FUNCTION_BLOCK FB_Cylinder EXTENDS FB_Component
VAR_INPUT
END_VAR
VAR_OUTPUT
END_VAR
VAR
	bInputA					AT%I*:		BOOL;
	bInputB					AT%I*:		BOOL;
	bOutputA				AT%Q*:		BOOL;
	bOutputB				AT%Q*:		BOOL;
	stSettings:				ST_CylinderSettings;
	fbDebounceA:			FB_Debounce;
	fbDebounceB:			FB_Debounce;	
	fbTimeout:				TON;
END_VAR

METHOD PUBLIC M_Cycle
VAR_INPUT
END_VAR
SUPER^.M_Cycle();

// Timeout
fbTimeout();
fbTimeout.IN:= FALSE;

// Debounc inputs
fbDebounceA(bInput:= bInputA);
fbDebounceB(bInput:= bInputB);
END_METHOD

METHOD PUBLIC M_Disable : BOOL
VAR_INPUT
END_VAR
bOutputA:= FALSE;
bOutputB:= FALSE;
M_Disable:= TRUE;
END_METHOD

METHOD PROTECTED M_Execute : BOOL // Return state complete
VAR_INPUT
END_VAR
IF M_HasMode(E_Mode.Manual) OR Globals.bSimulation THEN
	;
ELSE
	IF fbDebounceA.bValue AND fbDebounceB.bValue THEN
		P_Event.M_AddSTRING(P_Identifier);
		P_Event.M_AddSTRING(stSettings.sIdA);
		P_Event.M_AddSTRING(stSettings.sIdB);
		P_Event.M_Stop('Cylinder %s Logic error Inputs %s, %s are true', 0);
	END_IF	

	IF bOutputA THEN
		IF NOT fbDebounceA.bValue THEN
			fbTimeout.IN:= TRUE;
			IF fbTimeout.Q THEN
				P_Event.M_AddSTRING(P_Identifier);
				P_Event.M_AddSTRING(stSettings.sIdA);
				P_Event.M_Stop('Cylinder %s homeposition not reached %s', 0);				
			END_IF
		END_IF
	
	ELSIF bOutputB THEN
		IF NOT fbDebounceB.bValue THEN
			fbTimeout.IN:= TRUE;
			IF fbTimeout.Q THEN
				P_Event.M_AddSTRING(P_Identifier);
				P_Event.M_AddSTRING(stSettings.sIdB);
				P_Event.M_Stop('Cylinder %s workposition not reached %s', 0);				
			END_IF
		END_IF		
	END_IF
END_IF
END_METHOD

METHOD PROTECTED M_Starting : BOOL // Return state complete
VAR_INPUT
END_VAR
M_Starting:= SUPER^.M_Starting();

// Settings
fbTimeout.PT:= stSettings.tTimeout;
fbDebounceA.tTime:= stSettings.tDebounceA;
fbDebounceB.tTime:= stSettings.tDebounceB;
END_METHOD

METHOD PUBLIC M_ToHome : BOOL
VAR_INPUT
END_VAR
bOutputA:= TRUE;
bOutputB:= FALSE;
M_ToHome:= (bInputA AND NOT bInputB) OR Globals.bSimulation;
END_METHOD

METHOD PUBLIC M_ToWork : BOOL
VAR_INPUT
END_VAR
bOutputA:= FALSE;
bOutputB:= TRUE;
M_ToWork:= (bInputB AND NOT bInputA) OR Globals.bSimulation;
END_METHOD

PROPERTY PUBLIC P_Settings : REFERENCE TO ST_CylinderSettings
GET
P_Settings ref= stSettings;
END_GET
END_PROPERTY

END_FUNCTION_BLOCK

(* stored: Version 1.1.0.1
   POU FB_Cylinder: Id {0e789de7-7fe2-0204-3f8e-57ce5ee55d5b}, SpecialFunc None
   Method M_Cycle: Id {1e9e9c3d-3912-0fa8-3236-68f78e1ae73a}
   Method M_Disable: Id {084d4cc3-90c8-03fb-3f3b-46af82c7c547}
   Method M_Execute: Id {3442fc22-050d-094c-015a-424104d580c9}
   Method M_Starting: Id {be59c090-c9a2-0f0f-1926-c6952b267171}
   Method M_ToHome: Id {e25a0059-ac3f-0fc7-183d-9c8c2fedf38c}
   Method M_ToWork: Id {f6a4519f-a033-0321-07a0-e77d6b54d36a}
   Property P_Settings: Id {e36a7ccd-2016-0de5-3888-ff7d218b5f47}
   Get Get: Id {42d7fca6-98d0-0422-2538-b20afcaaa99e} *)
